// TIA Portal project "Project_v3_nuovo" (V15.1)

(* hardware
DEVICE "S7-1200 station_1"  S7-1200 Station
   slot 0: "Telaio di montaggio_0"  S7-1200 Rack  Rack  V1.0
   slot 1: "PLC_1"  CPU 1215C AC/DC/Rly  6ES7 215-1BG40-0XB0  V4.2
*)

// ===== PLC "PLC_1"  CPU 1215C AC/DC/Rly =====

VAR_GLOBAL   // PLC tag table "Tabella delle variabili standard"
   "GripperOpenStop" AT %I0.0 : Bool;
   "GripperCounter" AT %I0.1 : Bool;
   "ArmBackStop" AT %I0.2 : Bool;
   "ArmHCounter" AT %I0.3 : Bool;
   "ArmTopStop" AT %I0.4 : Bool;
   "ArmRotationStop" AT %I0.5 : Bool;
   "RotationalEncoder" AT %ID1000 : DInt;
   "VerticalEncoder" AT %ID1004 : DInt;
   "ConnectionButton" AT %I1.2 : Bool;
   "StopButton" AT %I1.3 : Bool;
   "ResetButton" AT %I1.4 : Bool;
   "In3" AT %I1.5 : Bool;
   "GripperOpen" AT %Q0.0 : Bool;
   "GripperClose" AT %Q0.1 : Bool;
   "ArmFront" AT %Q0.2 : Bool;
   "ArmBack" AT %Q0.3 : Bool;
   "ArmDown" AT %Q0.4 : Bool;
   "ArmUp" AT %Q0.5 : Bool;
   "RotationClockwise" AT %Q0.6 : Bool;
   "RotationCounterclockwise" AT %Q0.7 : Bool;
   "GreenLed" AT %Q1.0 : Bool;
   "RedLed" AT %Q1.1 : Bool;
   "System_Byte" AT %MB6 : Byte;
   "FirstScan" AT %M6.0 : Bool;
   "DiagStatusUpdate" AT %M6.1 : Bool;
   "AlwaysTRUE" AT %M6.2 : Bool;
   "AlwaysFALSE" AT %M6.3 : Bool;
   "RotationalCounter" AT %MW2 : UInt;
   "Clock_Byte" AT %MB0 : Byte;
   "Clock_10Hz" AT %M0.0 : Bool;
   "Clock_5Hz" AT %M0.1 : Bool;
   "Clock_2.5Hz" AT %M0.2 : Bool;
   "Clock_2Hz" AT %M0.3 : Bool;
   "Clock_1.25Hz" AT %M0.4 : Bool;
   "Clock_1Hz" AT %M0.5 : Bool;
   "Clock_0.625Hz" AT %M0.6 : Bool;
   "Clock_0.5Hz" AT %M0.7 : Bool;
   "VerticalCounter" AT %MW4 : UInt;
   "ForceReset" AT %M7.0 : Bool;
   "ResetCompleted" AT %M7.1 : Bool;
   "TCON_Req" AT %M1.0 : Bool;
   "TDIS_Req" AT %M1.1 : Bool;
   "TSEND_Req" AT %M1.2 : Bool;
   "TRCV_Req" AT %M1.3 : Bool;
   "VerticalOverCounter" AT %MW8 : Int;
   "VerticalUnderCounter" AT %MW10 : Int;
   "RotationOverCounter" AT %MW12 : Int;
   "RotationUnderCounter" AT %MW14 : Int;
   "NormalizedRotationUnderCounter" AT %MW16 : Int;
   "NormalizedVerticalUnderCounter" AT %MW18 : Int;
   "StopAll" AT %M20.1 : Bool;
   "HRegistered" AT %M20.2 : Bool;
   "RRegistered" AT %M20.3 : Bool;
   "VRegistered" AT %M20.4 : Bool;
END_VAR

DATA_BLOCK "Sent_values"   // DB10
{ S7_Optimized_Access := 'FALSE' }
VERSION : 0.1
   VAR
      Rotation : Int;
      Vertical : Int;
      Horizontal : Int;
      Gripper : Bool;
   END_VAR
BEGIN
END_DATA_BLOCK

DATA_BLOCK "Received_values"   // DB12
{ S7_Optimized_Access := 'FALSE' }
VERSION : 0.1
   VAR
      Rotation : Int;
      Vertical : Int;
      Horizontal : Int;
      Gripper : Bool;
   END_VAR
BEGIN
END_DATA_BLOCK

// folder: System blocks/Program resources

DATA_BLOCK "ArmHCounterCTUD"   // DB3
{ S7_Optimized_Access := 'TRUE' }
AUTHOR : Simatic
FAMILY : IEC
NAME : CNTR
VERSION : 1.0
// stored: InstanceOfName IEC_COUNTER
"IEC_COUNTER"
BEGIN
END_DATA_BLOCK

DATA_BLOCK "GripperStatus"   // DB4
{ S7_Optimized_Access := 'TRUE' }
AUTHOR : Simatic
FAMILY : IEC
NAME : CNTR
VERSION : 1.0
// stored: InstanceOfName IEC_COUNTER
"IEC_COUNTER"
BEGIN
END_DATA_BLOCK

DATA_BLOCK "GripperCounterCTUD"   // DB5
{ S7_Optimized_Access := 'TRUE' }
AUTHOR : Simatic
FAMILY : IEC
NAME : CNTR
VERSION : 1.0
// stored: InstanceOfName IEC_COUNTER
"IEC_COUNTER"
BEGIN
END_DATA_BLOCK

DATA_BLOCK "ArmHStatus"   // DB6
{ S7_Optimized_Access := 'TRUE' }
AUTHOR : Simatic
FAMILY : IEC
NAME : CNTR
VERSION : 1.0
// stored: InstanceOfName IEC_COUNTER
"IEC_COUNTER"
BEGIN
END_DATA_BLOCK

DATA_BLOCK "PLC_1_Connection_DB"   // DB7
{ S7_Optimized_Access := 'TRUE' }
AUTHOR : SIMATIC
FAMILY : MC7Plus
NAME : TC_IP_v4
VERSION : 1.0
// stored: InstanceOfName TCON_IP_v4
"TCON_IP_v4"
BEGIN
   ID := 1;
   InterfaceId := 64;
   RemotePort := 2000;
   ActiveEstablished := true;
   RemoteAddress.ADDR[1] := 192;
   RemoteAddress.ADDR[2] := 168;
   RemoteAddress.ADDR[4] := 241;
END_DATA_BLOCK

DATA_BLOCK "ArmHStatusCTUD"   // DB13
{ S7_Optimized_Access := 'TRUE' }
AUTHOR : Simatic
FAMILY : IEC
NAME : CNTR
VERSION : 1.0
// stored: InstanceOfName IEC_COUNTER
"IEC_COUNTER"
BEGIN
END_DATA_BLOCK

DATA_BLOCK "IEC_Timer_0_DB"   // DB14
{ S7_Optimized_Access := 'TRUE' }
AUTHOR : Simatic
FAMILY : IEC
NAME : IEC_TMR
VERSION : 1.0
// stored: InstanceOfName IEC_TIMER
"IEC_TIMER"
BEGIN
END_DATA_BLOCK

DATA_BLOCK "IEC_Timer_0_DB_1"   // DB15
{ S7_Optimized_Access := 'TRUE' }
AUTHOR : Simatic
FAMILY : IEC
NAME : IEC_TMR
VERSION : 1.0
// stored: InstanceOfName IEC_TIMER
"IEC_TIMER"
BEGIN
END_DATA_BLOCK

// folder: (top level)

ORGANIZATION_BLOCK "Main"   // OB1, LAD, ProgramCycle
TITLE = "Main Program Sweep (Cycle)"
{ S7_Optimized_Access := 'TRUE' }
VERSION : 0.1
   VAR_INPUT
      Initial_Call : Bool;   // Initial call of this OB
      Remanence : Bool;   // =True, if remanent data are available
   END_VAR
   VAR_TEMP   // added for the SCL form of the ladder/FBD networks
      _w1 : Bool;
      _w2 : Bool;
      _w3 : Bool;
   END_VAR
BEGIN

REGION Network 1
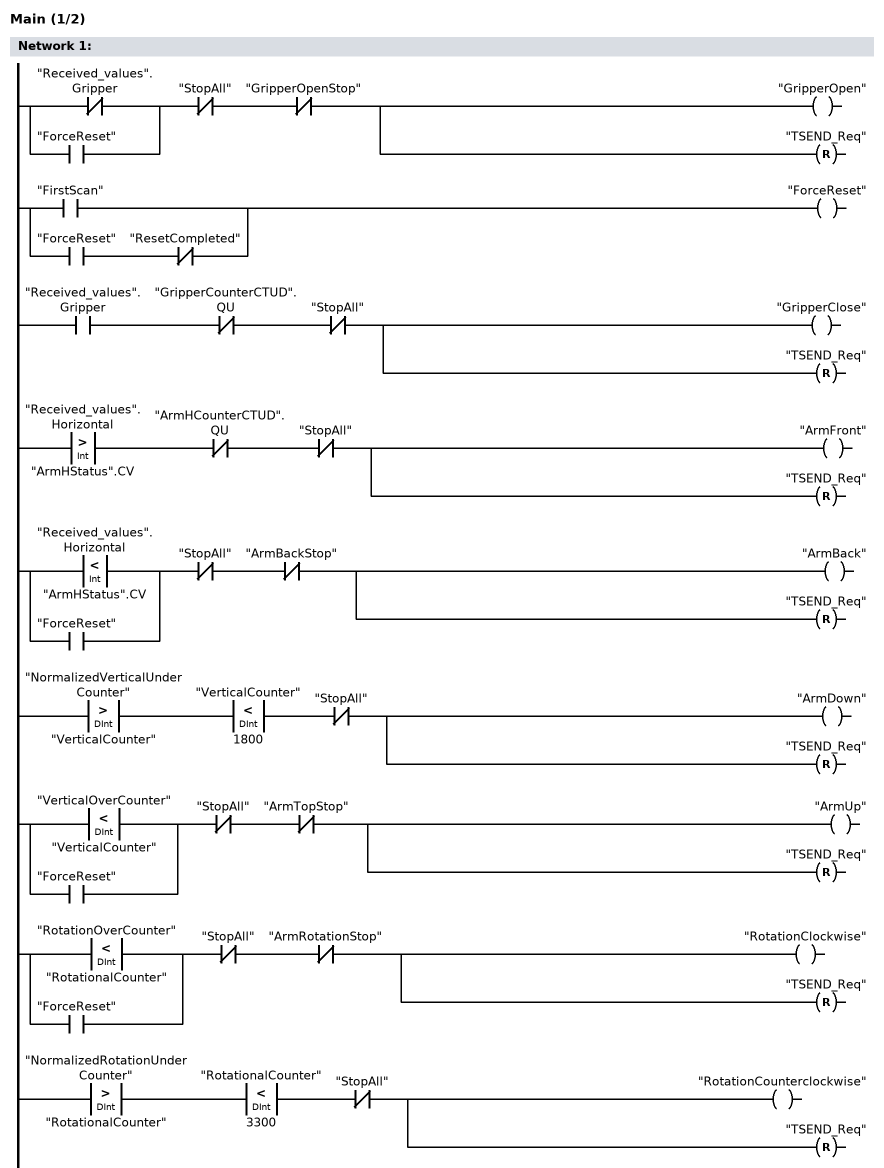
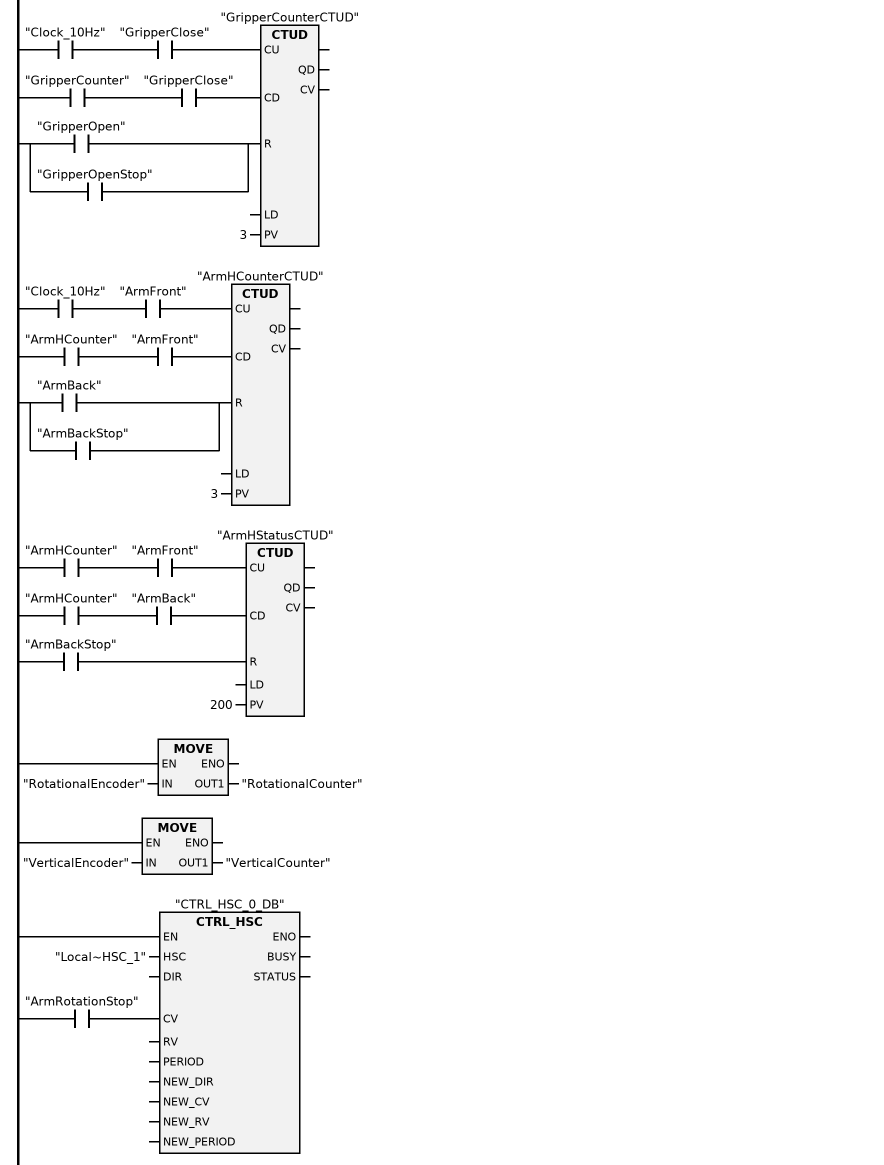
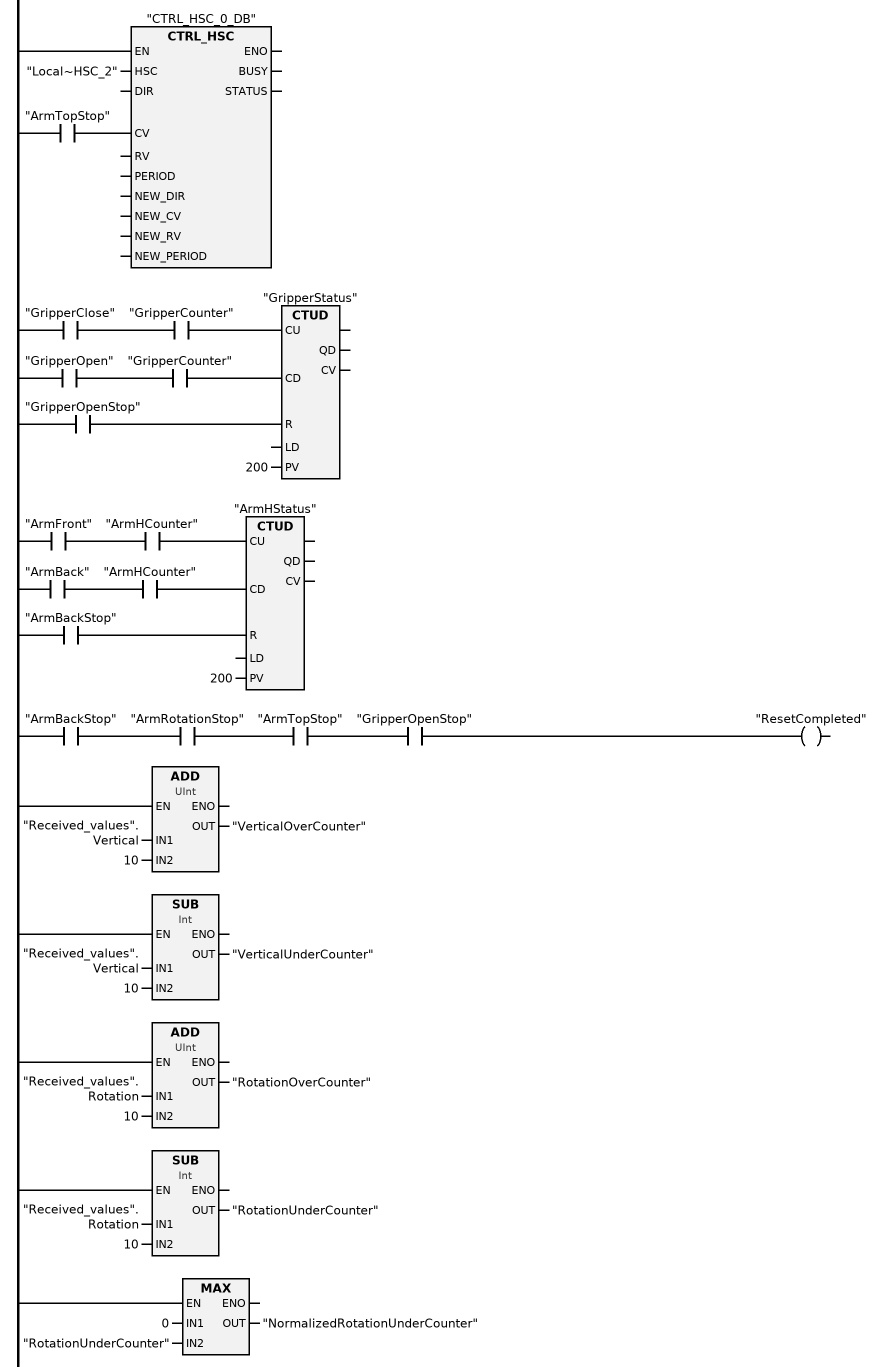
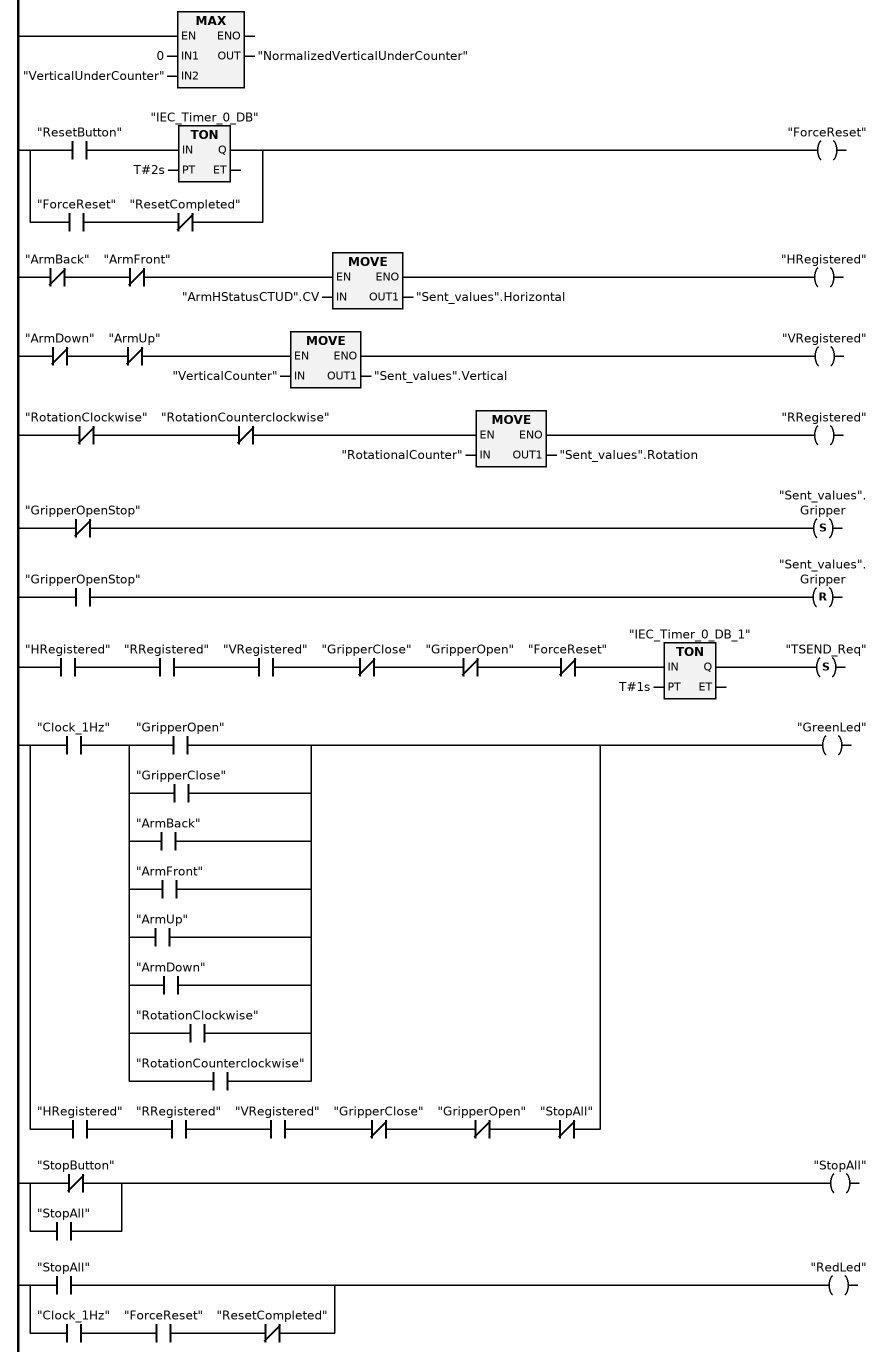
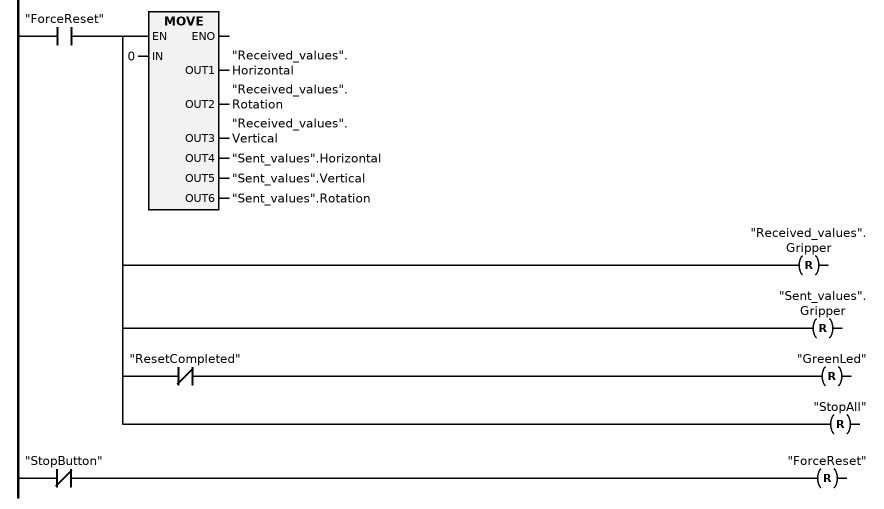
   "GripperOpen" := (NOT "Received_values".Gripper OR "ForceReset") AND NOT "StopAll" AND NOT "GripperOpenStop";
   IF "GripperOpen" THEN "TSEND_Req" := FALSE; END_IF;
   "ForceReset" := "FirstScan" OR ("ForceReset" AND NOT "ResetCompleted");
   "GripperClose" := "Received_values".Gripper AND NOT "GripperCounterCTUD".QU AND NOT "StopAll";
   IF "GripperClose" THEN "TSEND_Req" := FALSE; END_IF;
   "ArmFront" := ("Received_values".Horizontal > "ArmHStatus".CV) AND NOT "ArmHCounterCTUD".QU AND NOT "StopAll";
   IF "ArmFront" THEN "TSEND_Req" := FALSE; END_IF;
   "ArmBack" := (("Received_values".Horizontal < "ArmHStatus".CV) OR "ForceReset") AND NOT "StopAll" AND NOT "ArmBackStop";
   IF "ArmBack" THEN "TSEND_Req" := FALSE; END_IF;
   "ArmDown" := ("NormalizedVerticalUnderCounter" > "VerticalCounter") AND ("VerticalCounter" < 1800) AND NOT "StopAll";
   IF "ArmDown" THEN "TSEND_Req" := FALSE; END_IF;
   "ArmUp" := (("VerticalOverCounter" < "VerticalCounter") OR "ForceReset") AND NOT "StopAll" AND NOT "ArmTopStop";
   IF "ArmUp" THEN "TSEND_Req" := FALSE; END_IF;
   "RotationClockwise" := (("RotationOverCounter" < "RotationalCounter") OR "ForceReset") AND NOT "StopAll" AND NOT "ArmRotationStop";
   IF "RotationClockwise" THEN "TSEND_Req" := FALSE; END_IF;
   "RotationCounterclockwise" := ("NormalizedRotationUnderCounter" > "RotationalCounter") AND ("RotationalCounter" < 3300) AND NOT "StopAll";
   IF "RotationCounterclockwise" THEN "TSEND_Req" := FALSE; END_IF;
   "GripperCounterCTUD".CTUD(CU := "Clock_10Hz" AND "GripperClose",
                           CD := "GripperCounter" AND "GripperClose",
                           R := "GripperOpen" OR "GripperOpenStop",
                           PV := 3);
   "ArmHCounterCTUD".CTUD(CU := "Clock_10Hz" AND "ArmFront",
                          CD := "ArmHCounter" AND "ArmFront",
                          R := "ArmBack" OR "ArmBackStop",
                          PV := 3);
   "ArmHStatusCTUD".CTUD(CU := "ArmHCounter" AND "ArmFront",
                         CD := "ArmHCounter" AND "ArmBack",
                         R := "ArmBackStop",
                         PV := 200);
   "RotationalCounter" := "RotationalEncoder";
   "VerticalCounter" := "VerticalEncoder";
   "CTRL_HSC_0_DB"(HSC := "Local~HSC_1", CV := "ArmRotationStop");   // CTRL_HSC
   "CTRL_HSC_0_DB"(HSC := "Local~HSC_2", CV := "ArmTopStop");   // CTRL_HSC
   "GripperStatus".CTUD(CU := "GripperClose" AND "GripperCounter",
                        CD := "GripperOpen" AND "GripperCounter",
                        R := "GripperOpenStop",
                        PV := 200);
   "ArmHStatus".CTUD(CU := "ArmFront" AND "ArmHCounter",
                     CD := "ArmBack" AND "ArmHCounter",
                     R := "ArmBackStop",
                     PV := 200);
   "ResetCompleted" := "ArmBackStop" AND "ArmRotationStop" AND "ArmTopStop" AND "GripperOpenStop";
   "VerticalOverCounter" := "Received_values".Vertical + 10;
   "VerticalUnderCounter" := "Received_values".Vertical - 10;
   "RotationOverCounter" := "Received_values".Rotation + 10;
   "RotationUnderCounter" := "Received_values".Rotation - 10;
   "NormalizedRotationUnderCounter" := MAX(IN1 := 0, IN2 := "RotationUnderCounter");
   "NormalizedVerticalUnderCounter" := MAX(IN1 := 0, IN2 := "VerticalUnderCounter");
   "IEC_Timer_0_DB".TON(IN := "ResetButton", PT := T#2s);
   "ForceReset" := "IEC_Timer_0_DB".Q OR ("ForceReset" AND NOT "ResetCompleted");
   #_w1 := NOT "ArmBack" AND NOT "ArmFront";
   IF #_w1 THEN "Sent_values".Horizontal := "ArmHStatusCTUD".CV; END_IF;
   "HRegistered" := #_w1;
   #_w2 := NOT "ArmDown" AND NOT "ArmUp";
   IF #_w2 THEN "Sent_values".Vertical := "VerticalCounter"; END_IF;
   "VRegistered" := #_w2;
   #_w3 := NOT "RotationClockwise" AND NOT "RotationCounterclockwise";
   IF #_w3 THEN "Sent_values".Rotation := "RotationalCounter"; END_IF;
   "RRegistered" := #_w3;
   IF NOT "GripperOpenStop" THEN "Sent_values".Gripper := TRUE; END_IF;
   IF "GripperOpenStop" THEN "Sent_values".Gripper := FALSE; END_IF;
   "IEC_Timer_0_DB_1".TON(IN := "HRegistered" AND "RRegistered" AND "VRegistered" AND NOT "GripperClose" AND NOT "GripperOpen" AND NOT "ForceReset",
                          PT := T#1s);
   IF "IEC_Timer_0_DB_1".Q THEN "TSEND_Req" := TRUE; END_IF;
   "GreenLed" := ("Clock_1Hz" AND ("GripperOpen" OR "GripperClose" OR "ArmBack" OR "ArmFront" OR "ArmUp" OR "ArmDown" OR "RotationClockwise" OR "RotationCounterclockwise")) OR ("HRegistered" AND "RRegistered" AND "VRegistered" AND NOT "GripperClose" AND NOT "GripperOpen" AND NOT "StopAll");
   "StopAll" := NOT "StopButton" OR "StopAll";
   "RedLed" := "StopAll" OR ("Clock_1Hz" AND "ForceReset" AND NOT "ResetCompleted");
   IF "ForceReset" THEN
       "Received_values".Horizontal := 0;
       "Received_values".Rotation := 0;
       "Received_values".Vertical := 0;
       "Sent_values".Horizontal := 0;
       "Sent_values".Vertical := 0;
       "Sent_values".Rotation := 0;
       "Received_values".Gripper := FALSE;
       "Sent_values".Gripper := FALSE;
   END_IF;
   IF "ForceReset" AND NOT "ResetCompleted" THEN "GreenLed" := FALSE; END_IF;
   IF "ForceReset" THEN "StopAll" := FALSE; END_IF;
   IF NOT "StopButton" THEN "ForceReset" := FALSE; END_IF;
END_REGION

REGION Network 2
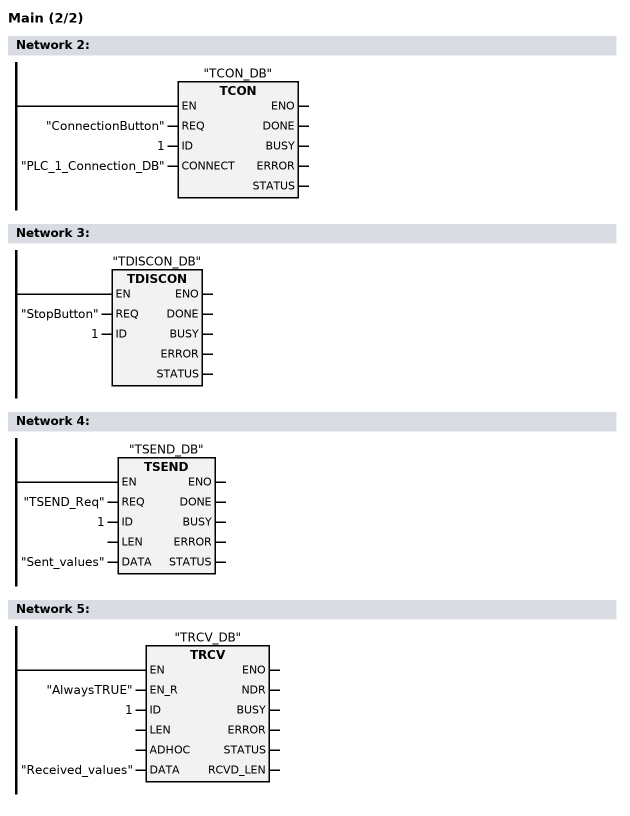
   "TCON_DB"(REQ := "ConnectionButton", ID := 1, CONNECT := "PLC_1_Connection_DB");   // TCON
END_REGION

REGION Network 3
   "TDISCON_DB"(REQ := "StopButton", ID := 1);   // TDISCON
END_REGION

REGION Network 4
   "TSEND_DB"(REQ := "TSEND_Req", ID := 1, DATA := "Sent_values");   // TSEND
END_REGION

REGION Network 5
   "TRCV_DB"(EN_R := "AlwaysTRUE", ID := 1, DATA := "Received_values");   // TRCV
END_REGION
END_ORGANIZATION_BLOCK